PROGRAM F_FIN_DUCHAS
VAR_INPUT
	Func:E_Funcio;
END_VAR
VAR
	///Activa
	xActv: BOOL;
	///Fin Funcion
	xFiFunc: BOOL;
	
	tFinDuchas: Ton;
END_VAR


(*Activa funcio *)
xActv:= func.Actv_Funcio;

tFinDuchas(IN:= xActv, PT:=T#5S);



(*FIN FUNCION*)
xFiFunc:=xActv AND NOT (tFinDuchas.Q);

END_PROGRAM

(* stored: Version 1.1.0.1, ProductVersion 3.1.4024.10
   POU F_FIN_DUCHAS: Id {99e8058a-e808-453f-b2e1-e553ff461907}, SpecialFunc None *)
